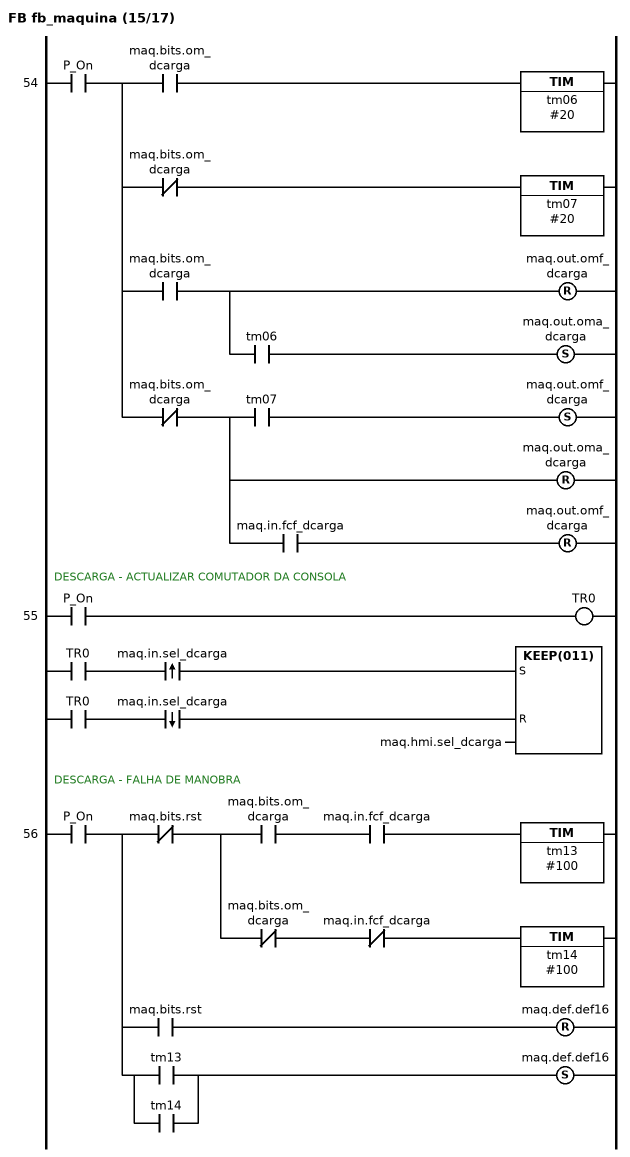
; rung 54
LD P_On
OUT TR0
AND maq.bits.om_dcarga
TIM tm06 #20
LD TR0
ANDNOT maq.bits.om_dcarga
TIM tm07 #20
LD TR0
AND maq.bits.om_dcarga
RSET maq.out.omf_dcarga
AND tm06
SET maq.out.oma_dcarga
LD TR0
ANDNOT maq.bits.om_dcarga
OUT TR1
AND tm07
SET maq.out.omf_dcarga
LD TR1
RSET maq.out.oma_dcarga
AND maq.in.fcf_dcarga
RSET maq.out.omf_dcarga
; rung 55: DESCARGA - ACTUALIZAR COMUTADOR DA CONSOLA
LD P_On
OUT TR0
LD TR0
@AND maq.in.sel_dcarga
LD TR0
%AND maq.in.sel_dcarga
KEEP(011) maq.hmi.sel_dcarga
; rung 56: DESCARGA - FALHA DE MANOBRA
LD P_On
OUT TR0
ANDNOT maq.bits.rst
OUT TR1
AND maq.bits.om_dcarga
AND maq.in.fcf_dcarga
TIM tm13 #100
LD TR1
ANDNOT maq.bits.om_dcarga
ANDNOT maq.in.fcf_dcarga
TIM tm14 #100
LD TR0
AND maq.bits.rst
RSET maq.def.def16
LD TR0
LD tm13
OR tm14
ANDLD
SET maq.def.def16

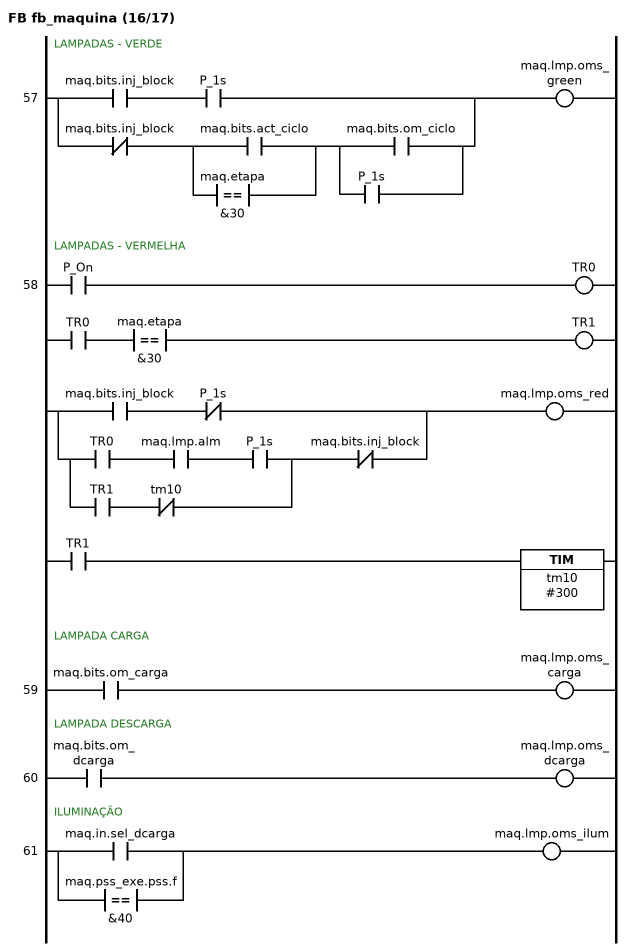
; rung 57: LAMPADAS - VERDE
LD maq.bits.inj_block
AND P_1s
LDNOT maq.bits.inj_block
LD maq.bits.act_ciclo
OR=(300) maq.etapa &30
ANDLD
LD maq.bits.om_ciclo
OR P_1s
ANDLD
ORLD
OUT maq.lmp.oms_green
; rung 58: LAMPADAS - VERMELHA
LD P_On
OUT TR0
LD TR0
AND=(300) maq.etapa &30
OUT TR1
LD maq.bits.inj_block
ANDNOT P_1s
LD TR0
AND maq.lmp.alm
AND P_1s
LD TR1
ANDNOT tm10
ORLD
ANDNOT maq.bits.inj_block
ORLD
OUT maq.lmp.oms_red
LD TR1
TIM tm10 #300
; rung 59: LAMPADA CARGA
LD maq.bits.om_carga
OUT maq.lmp.oms_carga
; rung 60: LAMPADA DESCARGA
LD maq.bits.om_dcarga
OUT maq.lmp.oms_dcarga
; rung 61: ILUMINAÇÃO
LD maq.in.sel_dcarga
OR=(300) maq.pss_exe.pss.f &40
OUT maq.lmp.oms_ilum

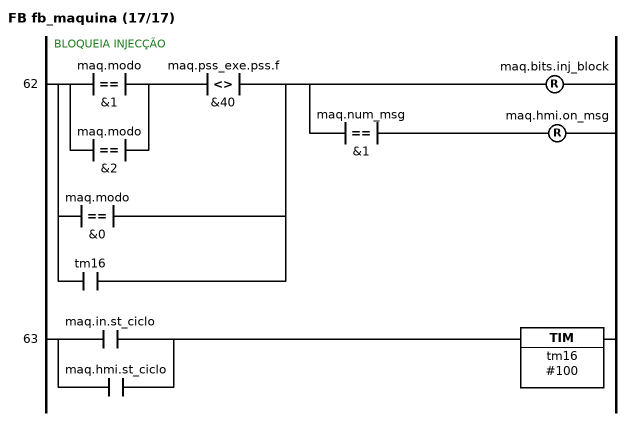
; rung 62: BLOQUEIA INJECÇÃO
LD=(300) maq.modo &1
OR=(300) maq.modo &2
AND<>(305) maq.pss_exe.pss.f &40
OR=(300) maq.modo &0
OR tm16
RSET maq.bits.inj_block
AND=(300) maq.num_msg &1
RSET maq.hmi.on_msg
; rung 63
LD maq.in.st_ciclo
OR maq.hmi.st_ciclo
TIM tm16 #100

## Function block fb_maquina_copy_log
; FUNÇÃO COPIA LOG - Copia os dados do passo actual para disponibilizar para fazer datalogger
VAR_INPUT
  tipo : INT;  (* Tipo de copia: 0 - Copia user/lote e dados a zero / 1 - Copia com ordem a decorrer (não copia user/lote) / 2 - Fim da ordem (Coloca passo 999) / 3 - Ordem descarregada sem execução (Colocar -3 no passo) *)
END_VAR
VAR_IN_OUT
  maq : s_maquina;  (* Dados da maquina *)
  of_exe : s_of;  (* Ordem de fabrico *)
  mes_com : s_mes_com;  (* Dados de comunicação com o MES *)
END_VAR
(*Não executa se ainda não tiver feito o log*)
IF maq.log.pss_exe.log=TRUE THEN
	RETURN;
END_IF;

maq.pss_exe.log:= TRUE;


(*Dados comuns*)
maq.log.user[0]:= mes_com.user[0];
maq.log.user[1]:= mes_com.user[1];
maq.log.user[2]:= mes_com.user[2];
maq.log.user[3]:= mes_com.user[3];
maq.log.user[4]:= mes_com.user[4];
maq.log.user[5]:= mes_com.user[5];
maq.log.user[6]:= mes_com.user[6];
maq.log.user[7]:= mes_com.user[7];
maq.log.user[8]:= mes_com.user[8];
maq.log.user[9]:= mes_com.user[9];
	
maq.log.n_of[0]:= of_exe.cliente.n_lt[0];
maq.log.n_of[1]:= of_exe.cliente.n_lt[1];
maq.log.n_of[2]:= of_exe.cliente.n_lt[2];
maq.log.n_of[3]:= of_exe.cliente.n_lt[3];
maq.log.n_of[4]:= of_exe.cliente.n_lt[4];
maq.log.n_of[5]:= of_exe.cliente.n_lt[5];
maq.log.n_of[6]:= of_exe.cliente.n_lt[6];
maq.log.n_of[7]:= of_exe.cliente.n_lt[7];
maq.log.n_of[8]:= of_exe.cliente.n_lt[8];
maq.log.n_of[9]:= of_exe.cliente.n_lt[9];

maq.log.pss_exe.exc:= maq.pss_exe.exc;
maq.log.pss_exe.exe:= maq.pss_exe.exe;	
maq.log.pss_exe.ini:= maq.pss_exe.ini;	
maq.log.pss_exe.fim:= maq.pss_exe.fim;	
maq.log.pss_exe.log:= maq.pss_exe.log;	

(*Registo inicial*)
IF tipo=0 THEN	
	maq.log.pss_exe.num_pss:= 0;
	maq.log.pss_exe.pss.f:= 0;
	maq.log.pss_exe.pss.p1:= 0;
	maq.log.pss_exe.pss.p2:= 0,0;
	maq.log.pss_exe.pss.tt:= 0,0;
	maq.log.pss_exe.pss.uni:= 0;
END_IF;

(*Ordem em execução*)
IF tipo=1 THEN	
	maq.log.pss_exe.num_pss:= maq.pss_exe.num_pss+1;
	maq.log.pss_exe.pss.f:= maq.pss_exe.pss.f;
	maq.log.pss_exe.pss.p1:= maq.pss_exe.pss.p1;
	maq.log.pss_exe.pss.p2:= maq.pss_exe.pss.p2;
	maq.log.pss_exe.pss.tt:= maq.pss_exe.pss.tt;
	maq.log.pss_exe.pss.uni:= maq.pss_exe.pss.uni;
END_IF;
	
(*Ordem terminada*)	
IF tipo=2 THEN
	maq.log.pss_exe.num_pss:= 999;
	maq.log.pss_exe.pss.f:= 0;
	maq.log.pss_exe.pss.p1:= 0;
	maq.log.pss_exe.pss.p2:= 0,0;
	maq.log.pss_exe.pss.tt:= 0,0;
	maq.log.pss_exe.pss.uni:= 0;
END_IF;	

(*Ordem não executada*)
IF tipo=3 THEN
	maq.log.pss_exe.num_pss:= -3;
	maq.log.pss_exe.pss.f:= 0;
	maq.log.pss_exe.pss.p1:= 0;
	maq.log.pss_exe.pss.p2:= 0,0;
	maq.log.pss_exe.pss.tt:= 0,0;
	maq.log.pss_exe.pss.uni:= 0;	
END_IF;	

## Function block fb_maquina_mov_pss_act
; FUNÇÃO MAQUINA MOVE PASSOS ACTUAIS - Faz a passagem da função do passo actual da maquina para a zona de memoria do passo actual. Faz também a passagem do total do passo em execução.
VAR_IN_OUT
  maq : s_maquina;  (* Dados da maquina *)
  of_exe : s_of;  (* Ordem de fabrico *)
END_VAR
(*Não esta a executar nenhum passo - Limpeza da zona de memória do passo actual*)
	IF maq.pss_exe.num_pss=-1 THEN
		maq.pss_exe.pss.f:= 0;
		maq.pss_exe.pss.p1:= 0;
		maq.pss_exe.pss.p2:=0,0;
		maq.pss_exe.pss.tt:= 0,0;
		maq.pss_exe.pss.uni:= 0;
	END_IF;

(*Leitura do passo actual e passagem dos valores*)
	IF maq.pss_exe.num_pss=0 THEN
		maq.pss_exe.pss.f:= of_exe.prg.pss[0].f;
		maq.pss_exe.pss.p1:= of_exe.prg.pss[0].p1;
		maq.pss_exe.pss.p2:= of_exe.prg.pss[0].p2;
		of_exe.prg.pss[0].tt:= maq.pss_exe.pss.tt;
		maq.pss_exe.pss.uni:=of_exe.prg.pss[0].uni;
	END_IF;

	IF maq.pss_exe.num_pss=1 THEN
		maq.pss_exe.pss.f:= of_exe.prg.pss[1].f;
		maq.pss_exe.pss.p1:= of_exe.prg.pss[1].p1;
		maq.pss_exe.pss.p2:= of_exe.prg.pss[1].p2;
		of_exe.prg.pss[1].tt:= maq.pss_exe.pss.tt;
		maq.pss_exe.pss.uni:=of_exe.prg.pss[1].uni;
	END_IF;

	IF maq.pss_exe.num_pss=2 THEN
		maq.pss_exe.pss.f:= of_exe.prg.pss[2].f;
		maq.pss_exe.pss.p1:= of_exe.prg.pss[2].p1;
		maq.pss_exe.pss.p2:= of_exe.prg.pss[2].p2;
		of_exe.prg.pss[2].tt:= maq.pss_exe.pss.tt;
		maq.pss_exe.pss.uni:=of_exe.prg.pss[2].uni;
	END_IF;

	IF maq.pss_exe.num_pss=3 THEN
		maq.pss_exe.pss.f:= of_exe.prg.pss[3].f;
		maq.pss_exe.pss.p1:= of_exe.prg.pss[3].p1;
		maq.pss_exe.pss.p2:= of_exe.prg.pss[3].p2;
		of_exe.prg.pss[3].tt:= maq.pss_exe.pss.tt;
		maq.pss_exe.pss.uni:=of_exe.prg.pss[3].uni;
	END_IF;

	IF maq.pss_exe.num_pss=4 THEN
		maq.pss_exe.pss.f:= of_exe.prg.pss[4].f;
		maq.pss_exe.pss.p1:= of_exe.prg.pss[4].p1;
		maq.pss_exe.pss.p2:= of_exe.prg.pss[4].p2;
		of_exe.prg.pss[4].tt:= maq.pss_exe.pss.tt;
		maq.pss_exe.pss.uni:=of_exe.prg.pss[4].uni;
	END_IF;

	IF maq.pss_exe.num_pss=5 THEN
		maq.pss_exe.pss.f:= of_exe.prg.pss[5].f;
		maq.pss_exe.pss.p1:= of_exe.prg.pss[5].p1;
		maq.pss_exe.pss.p2:= of_exe.prg.pss[5].p2;
		of_exe.prg.pss[5].tt:= maq.pss_exe.pss.tt;
		maq.pss_exe.pss.uni:=of_exe.prg.pss[5].uni;
	END_IF;

	IF maq.pss_exe.num_pss=6 THEN
		maq.pss_exe.pss.f:= of_exe.prg.pss[6].f;
		maq.pss_exe.pss.p1:= of_exe.prg.pss[6].p1;
		maq.pss_exe.pss.p2:= of_exe.prg.pss[6].p2;
		of_exe.prg.pss[6].tt:= maq.pss_exe.pss.tt;
		maq.pss_exe.pss.uni:=of_exe.prg.pss[6].uni;
	END_IF;

	IF maq.pss_exe.num_pss=7 THEN
		maq.pss_exe.pss.f:= of_exe.prg.pss[7].f;
		maq.pss_exe.pss.p1:= of_exe.prg.pss[7].p1;
		maq.pss_exe.pss.p2:= of_exe.prg.pss[7].p2;
		of_exe.prg.pss[7].tt:= maq.pss_exe.pss.tt;
		maq.pss_exe.pss.uni:=of_exe.prg.pss[7].uni;
	END_IF;

	IF maq.pss_exe.num_pss=8 THEN
		maq.pss_exe.pss.f:= of_exe.prg.pss[8].f;
		maq.pss_exe.pss.p1:= of_exe.prg.pss[8].p1;
		maq.pss_exe.pss.p2:= of_exe.prg.pss[8].p2;
		of_exe.prg.pss[8].tt:= maq.pss_exe.pss.tt;
		maq.pss_exe.pss.uni:=of_exe.prg.pss[8].uni;
	END_IF;

	IF maq.pss_exe.num_pss=9 THEN
		maq.pss_exe.pss.f:= of_exe.prg.pss[9].f;
		maq.pss_exe.pss.p1:= of_exe.prg.pss[9].p1;
		maq.pss_exe.pss.p2:= of_exe.prg.pss[9].p2;
		of_exe.prg.pss[9].tt:= maq.pss_exe.pss.tt;
		maq.pss_exe.pss.uni:=of_exe.prg.pss[9].uni;
	END_IF;

	IF maq.pss_exe.num_pss=10 THEN
		maq.pss_exe.pss.f:= of_exe.prg.pss[10].f;
		maq.pss_exe.pss.p1:= of_exe.prg.pss[10].p1;
		maq.pss_exe.pss.p2:= of_exe.prg.pss[10].p2;
		of_exe.prg.pss[10].tt:= maq.pss_exe.pss.tt;
		maq.pss_exe.pss.uni:=of_exe.prg.pss[10].uni;
	END_IF;

	IF maq.pss_exe.num_pss=11 THEN
		maq.pss_exe.pss.f:= of_exe.prg.pss[11].f;
		maq.pss_exe.pss.p1:= of_exe.prg.pss[11].p1;
		maq.pss_exe.pss.p2:= of_exe.prg.pss[11].p2;
		of_exe.prg.pss[11].tt:= maq.pss_exe.pss.tt;
		maq.pss_exe.pss.uni:=of_exe.prg.pss[11].uni;
	END_IF;

## Function block fb_maquina_pss_2_str10_PT
; FUNÇÃO PASSO PARA STRING - Transforma os passo em execução em strings para apresentar no HMI.
VAR_IN_OUT
  prg : s_of_prg;  (* Programa *)
  str_pss0 : STRING;  (* String do passo *)
  str_pss1 : STRING;  (* String do passo *)
  str_pss2 : STRING;  (* String do passo *)
  str_pss3 : STRING;  (* String do passo *)
  str_pss4 : STRING;  (* String do passo *)
  str_pss5 : STRING;  (* String do passo *)
  str_pss6 : STRING;  (* String do passo *)
  str_pss7 : STRING;  (* String do passo *)
  str_pss8 : STRING;  (* String do passo *)
  str_pss9 : STRING;  (* String do passo *)
  str_pss10 : STRING;
  str_pss11 : STRING;
  maq : s_maquina;  (* Dados da maquina *)
  str_act : STRING;  (* String do passo actual *)
END_VAR
VAR
  str_p1 : STRING;  (* Parametro 1 *)
  str_p2 : STRING;  (* Parametro 2 *)
  dd : REAL;  (* Dividendo *)
  dv : REAL;  (* Divisor *)
  qc : REAL;  (* Quociente *)
  r : REAL;  (* Resto *)
  i : INT;
  pss : s_of_pss;  (* Passo *)
  str_pss : STRING;  (* String do passo *)
END_VAR
FOR i:= 0 TO 11 DO
	(*Passagem dos dados dos varios passos*)
	CASE i OF
		0:	pss.f:= prg.pss[0].f;pss.p1:= prg.pss[0].p1;pss.p2:=prg.pss[0].p2;
		1:	pss.f:= prg.pss[1].f;pss.p1:= prg.pss[1].p1;pss.p2:=prg.pss[1].p2;
		2:	pss.f:= prg.pss[2].f;pss.p1:= prg.pss[2].p1;pss.p2:=prg.pss[2].p2;
		3:	pss.f:= prg.pss[3].f;pss.p1:= prg.pss[3].p1;pss.p2:=prg.pss[3].p2;
		4:	pss.f:= prg.pss[4].f;pss.p1:= prg.pss[4].p1;pss.p2:=prg.pss[4].p2;
		5:	pss.f:= prg.pss[5].f;pss.p1:= prg.pss[5].p1;pss.p2:=prg.pss[5].p2;
		6:	pss.f:= prg.pss[6].f;pss.p1:= prg.pss[6].p1;pss.p2:=prg.pss[6].p2;
		7:	pss.f:= prg.pss[7].f;pss.p1:= prg.pss[7].p1;pss.p2:=prg.pss[7].p2;
		8:	pss.f:= prg.pss[8].f;pss.p1:= prg.pss[8].p1;pss.p2:=prg.pss[8].p2;
		9:	pss.f:= prg.pss[9].f;pss.p1:= prg.pss[9].p1;pss.p2:=prg.pss[9].p2;
		10:	pss.f:= prg.pss[10].f;pss.p1:= prg.pss[10].p1;pss.p2:=prg.pss[10].p2;
		11:	pss.f:= prg.pss[11].f;pss.p1:= prg.pss[11].p1;pss.p2:=prg.pss[11].p2;
	END_CASE;
	(*Inicialização*)
		str_pss:= '';
 
 	(*Transformação dos valores em string*)
	 str_p1:= INT_TO_STRING(pss.p1);
 
 	dd:= pss.p2*10,0;
 	dv:= 10,0;
 	qc:=INT_TO_REAL(REAL_TO_INT(dd/dv));
 	r:= dd-dv*qc;
	IF r<0,0 THEN
		qc:= qc-1,0;
		r:= 10,0+r;
	END_IF;
	
 	str_p2:= CONCAT(INT_TO_STRING(REAL_TO_INT(qc)),',',INT_TO_STRING(REAL_TO_INT(r)));

  	(*Aspiração*)
 	IF pss.f=10 THEN
		 str_pss:=CONCAT('Aspirazione ',str_p1,'s');
	END_IF;

	(*Aquecimento*)
 	IF pss.f=20 THEN
		 str_pss:=CONCAT('Riscaldamento ',str_p2,'ºC ',str_p1,'s');
	END_IF;

  	(*Tratamento*)
 	IF pss.f=30 THEN
		 str_pss:=CONCAT('Trattamento ',str_p1,'s');
	END_IF;

  	(*Injecção*)
 	IF pss.f=40 THEN
		 CASE pss.p1 OF
		 	1:str_pss:=CONCAT('BOPSIL ',str_p2,'ml');  (*BOPSIL*)
			2:str_pss:=CONCAT('P28 ',str_p2,'ml');  (*P28*)
			3:str_pss:=CONCAT('SILBIONE ',str_p2,'ml');  (*SILICONE*)
			4:str_pss:=CONCAT('P2X ',str_p2,'ml');  (*P2X*)
			5:str_pss:=CONCAT('LC104 ',str_p2,'ml');  (*LC104*)
			6:str_pss:=CONCAT('PARAFFINA ',str_p2,'ml');  (*PARAFINA*)
			7:str_pss:=CONCAT('TEFLON ',str_p2,'ml');  (*TEFLON*)
			8:str_pss:=CONCAT('CAF ',str_p2,'ml');  (*CAF*)
			9:str_pss:=CONCAT('X15 ',str_p2,'ml');  (*X15*)
			10:str_pss:=CONCAT('SWAM P.N.S. ',str_p2,'ml');  (*SWAM P.N.S.*)
			11:str_pss:=CONCAT('SWAM P.SA ',str_p2,'ml');  (*SWAM P.SA*)		
			19:str_pss:=CONCAT('TR02 ',str_p2,'ml');  (*TR02*)
		END_CASE;
	END_IF;

  	(*LOAD*)
 	IF pss.f=70 THEN
		 str_pss:='Carico ';
	END_IF;

  	(*UNLOAD*)
 	IF pss.f=80 THEN
		 str_pss:='Scarico ';
	END_IF;
	
	(*Passagem das strings dos varios passos*)
	CASE i OF
		0:	str_pss0:= str_pss;
		1:	str_pss1:= str_pss;
		2:	str_pss2:= str_pss;
		3:	str_pss3:= str_pss;
		4:	str_pss4:= str_pss;
		5:	str_pss5:= str_pss;
		6:	str_pss6:= str_pss;
		7:	str_pss7:= str_pss;
		8:	str_pss8:= str_pss;
		9:	str_pss9:= str_pss;
		10:	str_pss10:= str_pss;
		11:	str_pss11:= str_pss;
	END_CASE;
	
	(*String do passo actual*)
	str_act:= '';
	CASE maq.pss_exe.num_pss OF
		0:	str_act:= str_pss0;
		1:	str_act:= str_pss1;
		2:	str_act:= str_pss2;
		3:	str_act:= str_pss3;
		4:	str_act:= str_pss4;
		5:	str_act:= str_pss5;
		6:	str_act:= str_pss6;
		7:	str_act:= str_pss7;
		8:	str_act:= str_pss8;
		9:	str_act:= str_pss9;
		10:	str_act:= str_pss10;
		11:	str_act:= str_pss11;
	END_CASE;
		
END_FOR;

## Function block fb_mes_com_exe
; COMUNICAÇÃO COM O MES - FUNÇÃO ARRANQUE DE ORDEM - Faz o controlo de comunicação do inicio de ordem com o MES
VAR_IN_OUT
  mes_com : s_mes_com;  (* Dados de comunicação com o MES *)
  of_exe : s_of;  (* Dados da ordem de fabrico a ser executada *)
END_VAR
VAR
  tm01 : TIMER;
  tm01_st : BOOL;
  mmss AT A351 : INT;
END_VAR
(*Falha de comunicação*)

tm01_st:=( mes_com.mes_plc =  mes_com.mes_plcx);
TIMX(tm01_st,tm01,600);
mes_com.mes_com_fail:= tm01.CF;

mes_com.mes_plcx:= mes_com.mes_plc;

(*Variável de comunicação para o MES*)
mes_com.plc_mes:= mmss;

(*FUNÇÕES
	0 - Nada
	1- Inicio de ordem
	2 - Fim de ordem
	3 - Cancela
	4 - Descarga sem tratamento
	*)
	
(*ESTADOS:
	0 - Nada
	1- Espera dados do MES
	2 - Inicio OK 
	3 - Fim OK
	4 - Erro de OF
	5 - Erro de user
	6 - Erro de comunicação*)

(* Função 0 - NADA*)

(* Função 1 - INICIO OF*)
IF mes_com.f_in_exe=1 AND (mes_com.ctrl_com_mes=0 OR mes_com.f_out_exe=1) THEN
	IF mes_com.f_out_exe=0 THEN

		mes_com.n_enc[0]:= of_exe.cliente.n_enc[0];
		mes_com.n_enc[1]:= of_exe.cliente.n_enc[1];
		mes_com.n_enc[2]:= of_exe.cliente.n_enc[2];
		mes_com.n_enc[3]:= of_exe.cliente.n_enc[3];
		mes_com.n_enc[4]:= of_exe.cliente.n_enc[4];
		mes_com.n_enc[5]:= of_exe.cliente.n_enc[5];
		mes_com.n_enc[6]:= of_exe.cliente.n_enc[6];
		mes_com.n_enc[7]:= of_exe.cliente.n_enc[7];
		mes_com.n_enc[8]:= of_exe.cliente.n_enc[8];
		mes_com.n_enc[9]:= of_exe.cliente.n_enc[9];

		mes_com.n_of[0]:= of_exe.cliente.n_of[0];
		mes_com.n_of[1]:= of_exe.cliente.n_of[1];
		mes_com.n_of[2]:= of_exe.cliente.n_of[2];
		mes_com.n_of[3]:= of_exe.cliente.n_of[3];
		mes_com.n_of[4]:= of_exe.cliente.n_of[4];
		mes_com.n_of[5]:= of_exe.cliente.n_of[5];
		mes_com.n_of[6]:= of_exe.cliente.n_of[6];
		mes_com.n_of[7]:= of_exe.cliente.n_of[7];
		mes_com.n_of[8]:= of_exe.cliente.n_of[8];
		mes_com.n_of[9]:= of_exe.cliente.n_of[9];		
		
		mes_com.n_lt[0]:= of_exe.cliente.n_lt[0];
		mes_com.n_lt[1]:= of_exe.cliente.n_lt[1];
		mes_com.n_lt[2]:= of_exe.cliente.n_lt[2];
		mes_com.n_lt[3]:= of_exe.cliente.n_lt[3];
		mes_com.n_lt[4]:= of_exe.cliente.n_lt[4];
		mes_com.n_lt[5]:= of_exe.cliente.n_lt[5];
		mes_com.n_lt[6]:= of_exe.cliente.n_lt[6];
		mes_com.n_lt[7]:= of_exe.cliente.n_lt[7];
		mes_com.n_lt[8]:= of_exe.cliente.n_lt[8];
		mes_com.n_lt[9]:= of_exe.cliente.n_lt[9];		
		
		mes_com.ctrl_com_plc:= -4;
		mes_com.new_of:= mes_com.new_of+1;
		IF mes_com.new_of>10000 OR mes_com.new_of<0 THEN
			mes_com.new_of:= 0;
		END_IF;		
	END_IF;
	mes_com.f_out_exe:= 1;
		(*MES OK - INICIO DE ORDEM*)
	IF mes_com.ctrl_com_mes=4 THEN
		mes_com.f_out_exe:= 2;
		 mes_com.f_in_exe:= 0;
		mes_com.ctrl_com_plc:= 0;		 
	END_IF;
		(*MES NOK - Mostra erro*)
	IF mes_com.ctrl_com_mes=101 THEN
		mes_com.f_out_exe:= 4;
		mes_com.f_in_exe:= 0;
		mes_com.ctrl_com_plc:= 0;		 
	END_IF;
	IF mes_com.ctrl_com_mes=102 THEN
		mes_com.f_out_exe:= 5;
		mes_com.f_in_exe:= 0;
		mes_com.ctrl_com_plc:= 0;		 
	END_IF;
END_IF;

(* Função 2 - FIM OF*)
IF mes_com.f_in_exe=2 THEN
	mes_com.ctrl_com_plc:= -5;	
	
	mes_com.f_out_exe:= 1;	
		(*MES OK - Ordem terminada*)
	IF mes_com.ctrl_com_mes=5 THEN
		mes_com.f_out_exe:= 3;
		 mes_com.f_in_exe:= 3;
		 mes_com.ctrl_com_plc:= 0;
	END_IF;
		(*MES NOK - Mostra erro*)
	IF mes_com.ctrl_com_mes=101 THEN
		mes_com.f_out_exe:= 4;
		mes_com.f_in_exe:= 3;
		mes_com.ctrl_com_plc:= 0;		 
	END_IF;
	IF mes_com.ctrl_com_mes=102 THEN
		mes_com.f_out_exe:= 5;
		mes_com.f_in_exe:= 3;
		mes_com.ctrl_com_plc:= 0;		 
	END_IF;	
END_IF;

(* Função 3 - CANCELA*)
IF mes_com.f_in_exe=3 THEN
	
	mes_com.ctrl_com_plc:= 0;
	mes_com.f_out_exe:= 0;
	mes_com.f_in_exe:= 0;
	
	mes_com.n_enc[0]:= 0;
	mes_com.n_enc[1]:= 0;
	mes_com.n_enc[2]:= 0;
	mes_com.n_enc[3]:= 0;
	mes_com.n_enc[4]:= 0;
	mes_com.n_enc[5]:= 0;
	mes_com.n_enc[6]:= 0;
	mes_com.n_enc[7]:= 0;
	mes_com.n_enc[8]:= 0;
	mes_com.n_enc[9]:= 0;
	
	mes_com.n_of[0]:= 0;
	mes_com.n_of[1]:= 0;
	mes_com.n_of[2]:= 0;
	mes_com.n_of[3]:= 0;
	mes_com.n_of[4]:= 0;
	mes_com.n_of[5]:= 0;
	mes_com.n_of[6]:= 0;
	mes_com.n_of[7]:= 0;
	mes_com.n_of[8]:= 0;
	mes_com.n_of[9]:= 0;
	
	mes_com.n_lt[0]:= 0;
	mes_com.n_lt[1]:= 0;
	mes_com.n_lt[2]:= 0;
	mes_com.n_lt[3]:= 0;
	mes_com.n_lt[4]:= 0;
	mes_com.n_lt[5]:= 0;
	mes_com.n_lt[6]:= 0;
	mes_com.n_lt[7]:= 0;
	mes_com.n_lt[8]:= 0;
	mes_com.n_lt[9]:= 0;	
		
END_IF;

(* Função 4 - DESCARGA SEM TRATAMENTO*)
IF mes_com.f_in_exe=4 THEN
		mes_com.ctrl_com_plc:= -3;

		mes_com.n_enc[0]:= of_exe.cliente.n_enc[0];
		mes_com.n_enc[1]:= of_exe.cliente.n_enc[1];
		mes_com.n_enc[2]:= of_exe.cliente.n_enc[2];
		mes_com.n_enc[3]:= of_exe.cliente.n_enc[3];
		mes_com.n_enc[4]:= of_exe.cliente.n_enc[4];
		mes_com.n_enc[5]:= of_exe.cliente.n_enc[5];
		mes_com.n_enc[6]:= of_exe.cliente.n_enc[6];
		mes_com.n_enc[7]:= of_exe.cliente.n_enc[7];
		mes_com.n_enc[8]:= of_exe.cliente.n_enc[8];
		mes_com.n_enc[9]:= of_exe.cliente.n_enc[9];

		mes_com.n_of[0]:= of_exe.cliente.n_of[0];
		mes_com.n_of[1]:= of_exe.cliente.n_of[1];
		mes_com.n_of[2]:= of_exe.cliente.n_of[2];
		mes_com.n_of[3]:= of_exe.cliente.n_of[3];
		mes_com.n_of[4]:= of_exe.cliente.n_of[4];
		mes_com.n_of[5]:= of_exe.cliente.n_of[5];
		mes_com.n_of[6]:= of_exe.cliente.n_of[6];
		mes_com.n_of[7]:= of_exe.cliente.n_of[7];
		mes_com.n_of[8]:= of_exe.cliente.n_of[8];
		mes_com.n_of[9]:= of_exe.cliente.n_of[9];		
		
		mes_com.n_lt[0]:= of_exe.cliente.n_lt[0];
		mes_com.n_lt[1]:= of_exe.cliente.n_lt[1];
		mes_com.n_lt[2]:= of_exe.cliente.n_lt[2];
		mes_com.n_lt[3]:= of_exe.cliente.n_lt[3];
		mes_com.n_lt[4]:= of_exe.cliente.n_lt[4];
		mes_com.n_lt[5]:= of_exe.cliente.n_lt[5];
		mes_com.n_lt[6]:= of_exe.cliente.n_lt[6];
		mes_com.n_lt[7]:= of_exe.cliente.n_lt[7];
		mes_com.n_lt[8]:= of_exe.cliente.n_lt[8];
		mes_com.n_lt[9]:= of_exe.cliente.n_lt[9];		
	
	mes_com.f_out_exe:= 1;	
		(*MES OK - Ordem terminada*)
	IF mes_com.ctrl_com_mes=3 THEN
		mes_com.f_out_exe:= 3;
		 mes_com.f_in_exe:= 3;
		 mes_com.ctrl_com_plc:= 0;
	END_IF;
		(*MES NOK - Mostra erro*)
	IF mes_com.ctrl_com_mes=101 THEN
		mes_com.f_out_exe:= 4;
		mes_com.f_in_exe:= 3;
		mes_com.ctrl_com_plc:= 0;		 
	END_IF;
	IF mes_com.ctrl_com_mes=102 THEN
		mes_com.f_out_exe:= 5;
		mes_com.f_in_exe:= 3;
		mes_com.ctrl_com_plc:= 0;		 
	END_IF;	
END_IF;
	
(*Falha de comunicação - Mostra janela de falha de comunicação*)
IF mes_com.mes_com_fail=TRUE THEN
	mes_com.f_out_exe:= 6;
	mes_com.f_in_exe:= 0;
	
	mes_com.ctrl_com_plc:= 0;
 	mes_com.ctrl_com_mes:= 0;		
END_IF;
IF  mes_com.mes_com_fail=FALSE AND mes_com.f_out_exe= 6 THEN
	mes_com.f_out_exe:= 0;
END_IF;

## Function block fb_mes_com_trp
; COMUNICAÇÃO COM O MES - FUNÇÃO TRANSPORTE - Faz o controlo de comunicação do transporte com o MES
VAR_INPUT
  ok_trp : BOOL;  (* Transporte OK *)
  ndp_trp : BOOL;  (* Transporte OK *)
END_VAR
VAR_IN_OUT
  mes_com : s_mes_com;  (* Dados de comunicação com o MES *)
  of_mes : s_of;  (* Dados da ordem de fabrico vindos do MES *)
  of_trp : s_of;  (* Dados da ordem de fabrico para o transporte *)
END_VAR
VAR
  tm01 : TIMER;
  tm02 : TIMER;
  tm01_st : BOOL;
  fb_of_clear : fb_of_clear;
  fb_of_copy : fb_of_copy;
  mmss AT A351 : INT;
  com_step : INT;
END_VAR
(*Falha de comunicação*)
tm01_st:=( mes_com.mes_plc =  mes_com.mes_plcx);
TIMX(tm01_st,tm01,600);
mes_com.mes_com_fail:= tm01.CF;

mes_com.mes_plcx:= mes_com.mes_plc;

(*Variável de comunicação para o MES*)
mes_com.plc_mes:= mmss;

(*FUNÇÕES
	0 - Nada
	1 - Pede info de OF
	2 - Transporta online
	3 - Cancela
	4 - Pede transporte offline
	5 - Transporta offline
	6 - Pede transporte online
	*)
	
(*ESTADOS:
	0 - Janela de introdução user/OF
	1 - Espera dados do MES
	2 - Janela de info de OF
	3 - Janela de transporte
	4 - Erro de OF
	5 - Erro de user
	6 - Erro de comunicação
	7 - Transporte manual
	8 - Transporte indisponivel
	9 - Maquina carregada
	10 - Ordem já alocada
	11 - Lote pertence à ordem actual*)

(* Função 0 - NADA*)

(* Função 1 - PEDE INFO DE OF*)
IF mes_com.f_in_exe=1 THEN
	IF com_step=0 AND  mes_com.ctrl_com_mes=0 THEN
		com_step:= 1;
	END_IF;
	
	IF com_step=1 THEN
		mes_com.ctrl_com_plc:= -1;
		mes_com.new_of:= mes_com.new_of+1;
		IF mes_com.new_of>10000 OR mes_com.new_of<0 THEN
			mes_com.new_of:= 0;
		END_IF;
		com_step:= 2;
	END_IF;
	mes_com.f_out_exe:= 1;
	IF com_step= 2 THEN
		(*MES OK - Mostra info da OF*)
		IF mes_com.ctrl_com_mes=1 THEN
			mes_com.f_out_exe:= 2;
			 mes_com.f_in_exe:= 0;
			 mes_com.ctrl_com_plc:= 0;
		END_IF;
			(*MES NOK - Mostra erro*)
		IF mes_com.ctrl_com_mes=101 THEN
			mes_com.f_out_exe:= 4;
			mes_com.f_in_exe:= 0;
			mes_com.ctrl_com_plc:= 0;
		END_IF;
		IF mes_com.ctrl_com_mes=102 THEN
			mes_com.f_out_exe:= 5;
			mes_com.f_in_exe:= 0;
			mes_com.ctrl_com_plc:= 0;
		END_IF;
		IF mes_com.ctrl_com_mes=103 THEN
			mes_com.f_out_exe:= 10;
			mes_com.f_in_exe:= 0;
			mes_com.ctrl_com_plc:= 0;
		END_IF;
		IF mes_com.ctrl_com_mes=104 THEN
			mes_com.f_out_exe:= 11;
			mes_com.f_in_exe:= 0;
			mes_com.ctrl_com_plc:= 0;
		END_IF;	
	END_IF;
END_IF;

(* Função 2 - TRANSPORTA*)
IF mes_com.f_in_exe=2 AND NOT of_trp.dados THEN
	IF mes_com.f_out_exe=2 THEN
		of_mes.dados:= TRUE;
		of_mes.online:= TRUE;
		fb_of_copy(of_mes,of_trp);
		mes_com.f_out_exe:= 3;
		 mes_com.f_in_exe:= 0;
		 mes_com.ctrl_com_plc:= 0;
	END_IF;	
END_IF;

(* Função 3 - CANCELA*)
IF mes_com.f_in_exe=3 THEN
	of_mes.dados:= FALSE;
	
	mes_com.ctrl_com_plc:= 0;
	com_step:= 0;
	mes_com.f_out_exe:= 0;
	mes_com.f_in_exe:= 0;
	
	mes_com.n_enc[0]:= 0;
	mes_com.n_enc[1]:= 0;
	mes_com.n_enc[2]:= 0;
	mes_com.n_enc[3]:= 0;
	mes_com.n_enc[4]:= 0;
	mes_com.n_enc[5]:= 0;
	mes_com.n_enc[6]:= 0;
	mes_com.n_enc[7]:= 0;
	mes_com.n_enc[8]:= 0;
	mes_com.n_enc[9]:= 0;
	
	mes_com.n_of[0]:= 0;
	mes_com.n_of[1]:= 0;
	mes_com.n_of[2]:= 0;
	mes_com.n_of[3]:= 0;
	mes_com.n_of[4]:= 0;
	mes_com.n_of[5]:= 0;
	mes_com.n_of[6]:= 0;
	mes_com.n_of[7]:= 0;
	mes_com.n_of[8]:= 0;
	mes_com.n_of[9]:= 0;
	
	mes_com.n_lt[0]:= 0;
	mes_com.n_lt[1]:= 0;
	mes_com.n_lt[2]:= 0;
	mes_com.n_lt[3]:= 0;
	mes_com.n_lt[4]:= 0;
	mes_com.n_lt[5]:= 0;
	mes_com.n_lt[6]:= 0;
	mes_com.n_lt[7]:= 0;
	mes_com.n_lt[8]:= 0;
	mes_com.n_lt[9]:= 0;	
	
	mes_com.user[0]:= 0;
	mes_com.user[1]:= 0;
	mes_com.user[2]:= 0;
	mes_com.user[3]:= 0;
	mes_com.user[4]:= 0;
	mes_com.user[5]:= 0;
	mes_com.user[6]:= 0;
	mes_com.user[7]:= 0;
	mes_com.user[8]:= 0;
	mes_com.user[9]:= 0;		
END_IF;

(*Pede transporte offline*)
IF mes_com.f_in_exe=4 THEN
	mes_com.f_out_exe:= 7;
	mes_com.f_in_exe:= 0;
	mes_com.ctrl_com_plc:= 0;	
END_IF;

(*Transporta offline*)
IF mes_com.f_in_exe=5 AND NOT of_trp.dados THEN
	of_mes.cliente.n_enc[0]:=  mes_com.n_enc[0];
	of_mes.cliente.n_enc[1]:=  mes_com.n_enc[1];
	of_mes.cliente.n_enc[2]:=  mes_com.n_enc[2];
	of_mes.cliente.n_enc[3]:=  mes_com.n_enc[3];
	of_mes.cliente.n_enc[4]:=  mes_com.n_enc[4];
	of_mes.cliente.n_enc[5]:=  mes_com.n_enc[5];
	of_mes.cliente.n_enc[6]:=  mes_com.n_enc[6];
	of_mes.cliente.n_enc[7]:=  mes_com.n_enc[7];
	of_mes.cliente.n_enc[8]:=  mes_com.n_enc[8];
	of_mes.cliente.n_enc[9]:=  mes_com.n_enc[9];
	
	of_mes.cliente.n_of[0]:=  mes_com.n_of[0];
	of_mes.cliente.n_of[1]:=  mes_com.n_of[1];
	of_mes.cliente.n_of[2]:=  mes_com.n_of[2];
	of_mes.cliente.n_of[3]:=  mes_com.n_of[3];
	of_mes.cliente.n_of[4]:=  mes_com.n_of[4];
	of_mes.cliente.n_of[5]:=  mes_com.n_of[5];
	of_mes.cliente.n_of[6]:=  mes_com.n_of[6];
	of_mes.cliente.n_of[7]:=  mes_com.n_of[7];
	of_mes.cliente.n_of[8]:=  mes_com.n_of[8];
	of_mes.cliente.n_of[9]:=  mes_com.n_of[9];
	
	of_mes.cliente.n_lt[0]:=  mes_com.n_lt[0];
	of_mes.cliente.n_lt[1]:=  mes_com.n_lt[1];
	of_mes.cliente.n_lt[2]:=  mes_com.n_lt[2];
	of_mes.cliente.n_lt[3]:=  mes_com.n_lt[3];
	of_mes.cliente.n_lt[4]:=  mes_com.n_lt[4];
	of_mes.cliente.n_lt[5]:=  mes_com.n_lt[5];
	of_mes.cliente.n_lt[6]:=  mes_com.n_lt[6];
	of_mes.cliente.n_lt[7]:=  mes_com.n_lt[7];
	of_mes.cliente.n_lt[8]:=  mes_com.n_lt[8];
	of_mes.cliente.n_lt[9]:=  mes_com.n_lt[9];	
	
	of_mes.dados:= TRUE;
	of_mes.online:= TRUE;
	fb_of_copy(of_mes,of_trp);
	mes_com.f_out_exe:= 3;
	 mes_com.f_in_exe:= 0;
	 mes_com.ctrl_com_plc:= 0;
END_IF;
	
(*Pede transporte online*)
IF mes_com.f_in_exe=6 THEN
	mes_com.f_out_exe:= 0;
	mes_com.f_in_exe:= 0;
	mes_com.ctrl_com_plc:= 0;
END_IF;	
	
IF  mes_com.mes_com_fail=FALSE AND mes_com.f_out_exe= 6 THEN
	mes_com.f_out_exe:= 0;
END_IF;

(*Transporte indisponivel*)
IF ok_trp=FALSE AND ( mes_com.f_out_exe= 0 OR  mes_com.f_out_exe= 7) THEN
	mes_com.f_out_exe:= 8;
	mes_com.f_in_exe:= 0;
END_IF;

IF ok_trp=TRUE AND mes_com.f_out_exe=8 THEN
	mes_com.f_out_exe:= 0;
END_IF;

(*Maquina carregada*)
IF of_trp.dados=TRUE AND ( mes_com.f_out_exe= 0 OR  mes_com.f_out_exe= 7) THEN
	mes_com.f_out_exe:= 9;
	mes_com.f_in_exe:= 0;
END_IF;
IF of_trp.dados=FALSE AND mes_com.f_out_exe=9 THEN
	mes_com.f_out_exe:= 0;
END_IF;

(*Transporte indisponivel*)
IF ndp_trp=TRUE AND ( mes_com.f_out_exe= 0 OR  mes_com.f_out_exe= 7) THEN
	mes_com.f_out_exe:= 12;
	mes_com.f_in_exe:= 0;
END_IF;

IF ndp_trp=FALSE AND mes_com.f_out_exe=12 THEN
	mes_com.f_out_exe:= 0;
END_IF;

(*Falha de comunicação - Mostra janela de falha de comunicação*)
IF mes_com.mes_com_fail=TRUE AND ( mes_com.f_out_exe=0  OR mes_com.f_out_exe=1) THEN
	mes_com.f_out_exe:= 6;
	mes_com.f_in_exe:= 0;
	
	mes_com.ctrl_com_plc:= 0;
 	mes_com.ctrl_com_mes:= 0;			
END_IF;
		
(*Termina ordem de transporte*)
IF mes_com.f_out_exe=3 and ndp_trp=TRUE THEN
	mes_com.f_in_exe:= 3;
END_IF;	

(*Novo pedido*)
IF mes_com.ctrl_com_plc=0 THEN
	com_step:= 0;
END_IF;

## Function block fb_mes_cparagem
; CAUSAS DE PARAGEM - Causas de paragem para o MES
VAR_IN_OUT
  maq : s_maquina;  (* Dados da maquina *)
END_VAR

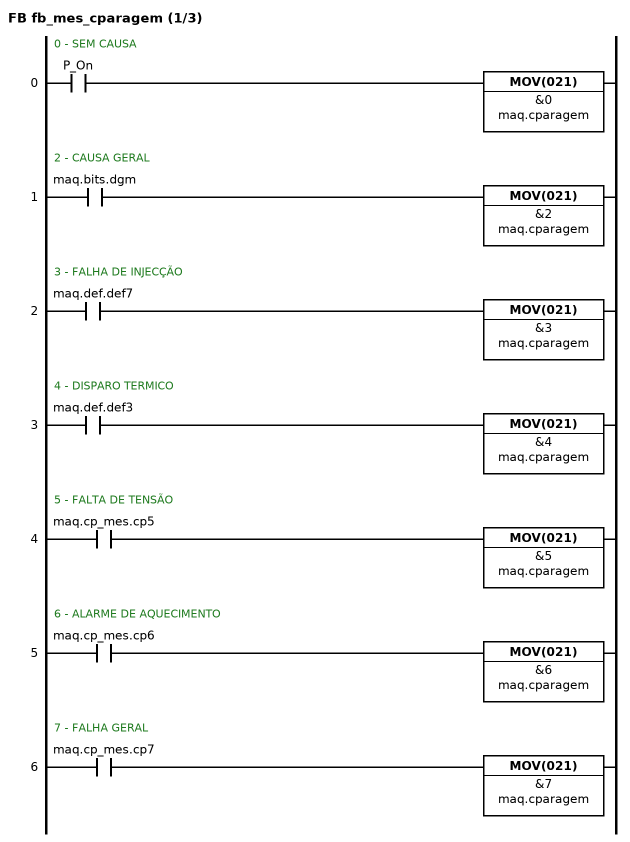
; rung 0: 0 - SEM CAUSA
LD P_On
MOV(021) &0 maq.cparagem
; rung 1: 2 - CAUSA GERAL
LD maq.bits.dgm
MOV(021) &2 maq.cparagem
; rung 2: 3 - FALHA DE INJECÇÃO
LD maq.def.def7
MOV(021) &3 maq.cparagem
; rung 3: 4 - DISPARO TERMICO
LD maq.def.def3
MOV(021) &4 maq.cparagem
; rung 4: 5 - FALTA DE TENSÃO
LD maq.cp_mes.cp5
MOV(021) &5 maq.cparagem
; rung 5: 6 - ALARME DE AQUECIMENTO
LD maq.cp_mes.cp6
MOV(021) &6 maq.cparagem
; rung 6: 7 - FALHA GERAL
LD maq.cp_mes.cp7
MOV(021) &7 maq.cparagem

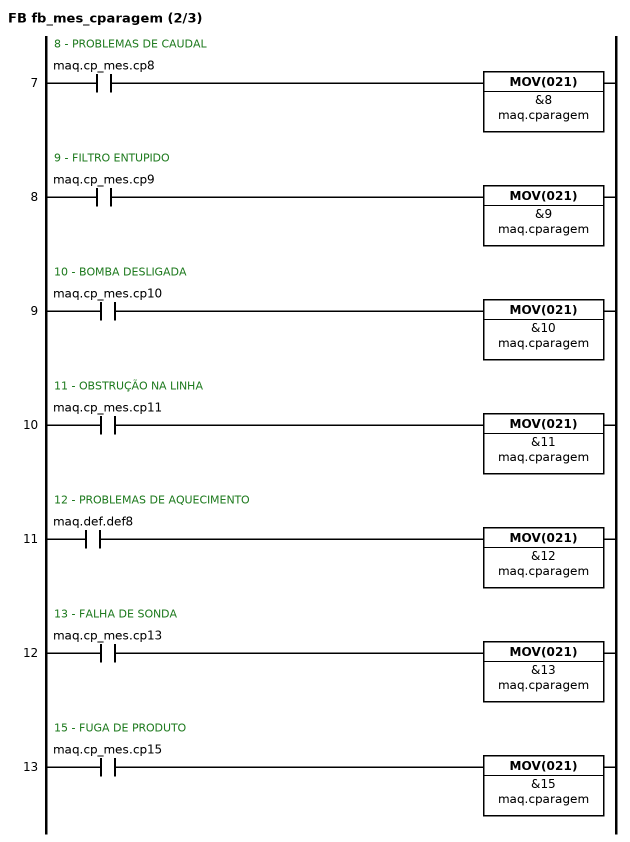
; rung 7: 8 - PROBLEMAS DE CAUDAL
LD maq.cp_mes.cp8
MOV(021) &8 maq.cparagem
; rung 8: 9 - FILTRO ENTUPIDO
LD maq.cp_mes.cp9
MOV(021) &9 maq.cparagem
; rung 9: 10 - BOMBA DESLIGADA
LD maq.cp_mes.cp10
MOV(021) &10 maq.cparagem
; rung 10: 11 - OBSTRUÇÃO NA LINHA
LD maq.cp_mes.cp11
MOV(021) &11 maq.cparagem
; rung 11: 12 - PROBLEMAS DE AQUECIMENTO
LD maq.def.def8
MOV(021) &12 maq.cparagem
; rung 12: 13 - FALHA DE SONDA
LD maq.cp_mes.cp13
MOV(021) &13 maq.cparagem
; rung 13: 15 - FUGA DE PRODUTO
LD maq.cp_mes.cp15
MOV(021) &15 maq.cparagem

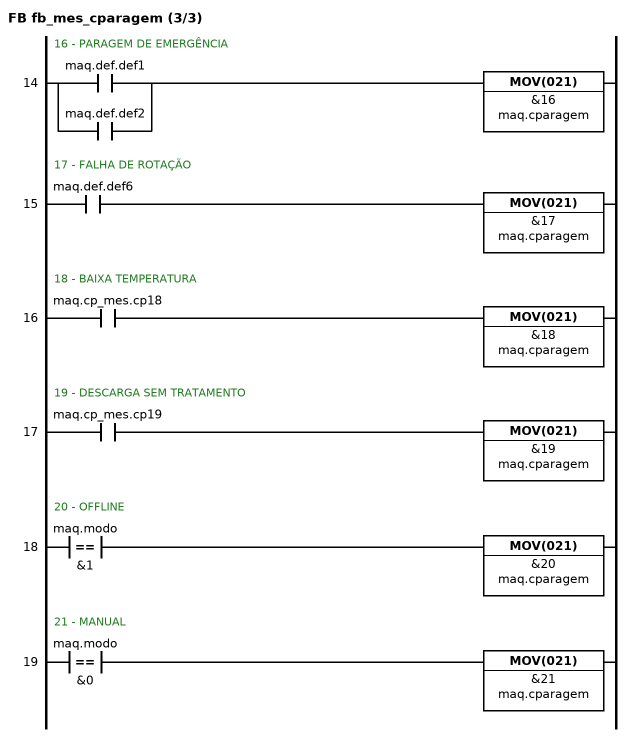
; rung 14: 16 - PARAGEM DE EMERGÊNCIA
LD maq.def.def1
OR maq.def.def2
MOV(021) &16 maq.cparagem
; rung 15: 17 - FALHA DE ROTAÇÃO
LD maq.def.def6
MOV(021) &17 maq.cparagem
; rung 16: 18 - BAIXA TEMPERATURA
LD maq.cp_mes.cp18
MOV(021) &18 maq.cparagem
; rung 17: 19 - DESCARGA SEM TRATAMENTO
LD maq.cp_mes.cp19
MOV(021) &19 maq.cparagem
; rung 18: 20 - OFFLINE
LD=(300) maq.modo &1
MOV(021) &20 maq.cparagem
; rung 19: 21 - MANUAL
LD=(300) maq.modo &0
MOV(021) &21 maq.cparagem

## Function block fb_of_clear
; FUNÇÃO LIMPA UMA ORDEM DE FABRICO - Coloca os valores da OF a zero.
VAR_IN_OUT
  of_in_out : s_of;  (* OF a ser apagada *)
END_VAR
(*Apaga uma OF*)
of_in_out.dados:= FALSE;

(*Cliente*)
of_in_out.cliente.nome[0]:=0;
of_in_out.cliente.nome[1]:=0;
of_in_out.cliente.nome[2]:=0;
of_in_out.cliente.nome[3]:=0;
of_in_out.cliente.nome[4]:=0;
of_in_out.cliente.nome[5]:=0;
of_in_out.cliente.nome[6]:=0;
of_in_out.cliente.nome[7]:=0;
of_in_out.cliente.nome[8]:=0;
of_in_out.cliente.nome[9]:=0;
of_in_out.cliente.nome[10]:=0;
of_in_out.cliente.nome[11]:=0;
of_in_out.cliente.nome[12]:=0;
of_in_out.cliente.nome[13]:=0;
of_in_out.cliente.nome[14]:=0;
of_in_out.cliente.nome[15]:=0;
of_in_out.cliente.nome[16]:=0;
of_in_out.cliente.nome[17]:=0;
of_in_out.cliente.nome[18]:=0;
of_in_out.cliente.nome[19]:=0;
of_in_out.cliente.nome[20]:=0;
of_in_out.cliente.nome[21]:=0;
of_in_out.cliente.nome[22]:=0;
of_in_out.cliente.nome[23]:=0;
of_in_out.cliente.nome[24]:=0;

of_in_out.cliente.data[0]:=0;
of_in_out.cliente.data[1]:=0;
of_in_out.cliente.data[2]:=0;
of_in_out.cliente.data[3]:=0;
of_in_out.cliente.data[4]:=0;
of_in_out.cliente.data[5]:=0;
of_in_out.cliente.data[6]:=0;
of_in_out.cliente.data[7]:=0;
of_in_out.cliente.data[8]:=0;
of_in_out.cliente.data[9]:=0;

of_in_out.cliente.produto[0]:=0;
of_in_out.cliente.produto[1]:=0;
of_in_out.cliente.produto[2]:=0;
of_in_out.cliente.produto[3]:=0;
of_in_out.cliente.produto[4]:=0;
of_in_out.cliente.produto[5]:=0;
of_in_out.cliente.produto[6]:=0;
of_in_out.cliente.produto[7]:=0;
of_in_out.cliente.produto[8]:=0;
of_in_out.cliente.produto[9]:=0;
of_in_out.cliente.produto[10]:=0;
of_in_out.cliente.produto[11]:=0;
of_in_out.cliente.produto[12]:=0;
of_in_out.cliente.produto[13]:=0;
of_in_out.cliente.produto[14]:=0;
of_in_out.cliente.produto[15]:=0;
of_in_out.cliente.produto[16]:=0;
of_in_out.cliente.produto[17]:=0;
of_in_out.cliente.produto[18]:=0;
of_in_out.cliente.produto[19]:=0;

of_in_out.cliente.prg_on[0]:=0;
of_in_out.cliente.prg_on[1]:=0;
of_in_out.cliente.prg_on[2]:=0;
of_in_out.cliente.prg_on[3]:=0;
of_in_out.cliente.prg_on[4]:=0;

of_in_out.cliente.n_enc[0]:=0;
of_in_out.cliente.n_enc[1]:=0;
of_in_out.cliente.n_enc[2]:=0;
of_in_out.cliente.n_enc[3]:=0;
of_in_out.cliente.n_enc[4]:=0;
of_in_out.cliente.n_enc[5]:=0;
of_in_out.cliente.n_enc[6]:=0;
of_in_out.cliente.n_enc[7]:=0;
of_in_out.cliente.n_enc[8]:=0;
of_in_out.cliente.n_enc[9]:=0;

of_in_out.cliente.n_of[0]:=0;
of_in_out.cliente.n_of[1]:=0;
of_in_out.cliente.n_of[2]:=0;
of_in_out.cliente.n_of[3]:=0;
of_in_out.cliente.n_of[4]:=0;
of_in_out.cliente.n_of[5]:=0;
of_in_out.cliente.n_of[6]:=0;
of_in_out.cliente.n_of[7]:=0;
of_in_out.cliente.n_of[8]:=0;
of_in_out.cliente.n_of[9]:=0;

of_in_out.cliente.n_lt[0]:=0;
of_in_out.cliente.n_lt[1]:=0;
of_in_out.cliente.n_lt[2]:=0;
of_in_out.cliente.n_lt[3]:=0;
of_in_out.cliente.n_lt[4]:=0;
of_in_out.cliente.n_lt[5]:=0;
of_in_out.cliente.n_lt[6]:=0;
of_in_out.cliente.n_lt[7]:=0;
of_in_out.cliente.n_lt[8]:=0;
of_in_out.cliente.n_lt[9]:=0;

(*Totais*)
of_in_out.totais.tt_global:=0;
of_in_out.totais.tt_falta:=0;
of_in_out.totais.tt_produzir:=0;

(*Calibre*)
of_in_out.calibre.dmt1:=0,0;
of_in_out.calibre.dmt2:=0,0;
of_in_out.calibre.h:=0,0;
of_in_out.calibre.a:=0,0;
of_in_out.calibre.qtp:=0,0;

of_in_out.calibre.cl_txt[0]:=0;
of_in_out.calibre.cl_txt[1]:=0;
of_in_out.calibre.cl_txt[2]:=0;
of_in_out.calibre.cl_txt[3]:=0;
of_in_out.calibre.cl_txt[4]:=0;
of_in_out.calibre.cl_txt[5]:=0;
of_in_out.calibre.cl_txt[6]:=0;
of_in_out.calibre.cl_txt[7]:=0;
of_in_out.calibre.cl_txt[8]:=0;
of_in_out.calibre.cl_txt[9]:=0;

(*Programa*)
of_in_out.prg.pss[0].f:=0;
of_in_out.prg.pss[0].p1:=0;
of_in_out.prg.pss[0].p2:=0,0;
of_in_out.prg.pss[0].tt:=0,0;
of_in_out.prg.pss[0].uni:=0;
of_in_out.prg.pss[0].uni:=12;
CASE of_in_out.prg.pss[0].f OF
	40:of_in_out.prg.pss[0].uni:=9;
END_CASE;

of_in_out.prg.pss[1].f:=0;
of_in_out.prg.pss[1].p1:=0;
of_in_out.prg.pss[1].p2:=0,0;
of_in_out.prg.pss[1].tt:=0,0;
of_in_out.prg.pss[1].uni:=0;
of_in_out.prg.pss[1].uni:=12;
CASE of_in_out.prg.pss[1].f OF
	40:of_in_out.prg.pss[1].uni:=9;
END_CASE;

of_in_out.prg.pss[2].f:=0;
of_in_out.prg.pss[2].p1:=0;
of_in_out.prg.pss[2].p2:=0,0;
of_in_out.prg.pss[2].tt:=0,0;
of_in_out.prg.pss[2].uni:=0;
of_in_out.prg.pss[2].uni:=12;
CASE of_in_out.prg.pss[2].f OF
	40:of_in_out.prg.pss[2].uni:=9;
END_CASE;

of_in_out.prg.pss[3].f:=0;
of_in_out.prg.pss[3].p1:=0;
of_in_out.prg.pss[3].p2:=0,0;
of_in_out.prg.pss[3].tt:=0,0;
of_in_out.prg.pss[3].uni:=0;
of_in_out.prg.pss[3].uni:=12;
CASE of_in_out.prg.pss[3].f OF
	40:of_in_out.prg.pss[3].uni:=9;
END_CASE;

of_in_out.prg.pss[4].f:=0;
of_in_out.prg.pss[4].p1:=0;
of_in_out.prg.pss[4].p2:=0,0;
of_in_out.prg.pss[4].tt:=0,0;
of_in_out.prg.pss[4].uni:=0;
of_in_out.prg.pss[4].uni:=12;
CASE of_in_out.prg.pss[4].f OF
	40:of_in_out.prg.pss[4].uni:=9;
END_CASE;

of_in_out.prg.pss[5].f:=0;
of_in_out.prg.pss[5].p1:=0;
of_in_out.prg.pss[5].p2:=0,0;
of_in_out.prg.pss[5].tt:=0,0;
of_in_out.prg.pss[5].uni:=0;
of_in_out.prg.pss[5].uni:=12;
CASE of_in_out.prg.pss[5].f OF
	40:of_in_out.prg.pss[5].uni:=9;
END_CASE;

of_in_out.prg.pss[6].f:=0;
of_in_out.prg.pss[6].p1:=0;
of_in_out.prg.pss[6].p2:=0,0;
of_in_out.prg.pss[6].tt:=0,0;
of_in_out.prg.pss[6].uni:=0;
of_in_out.prg.pss[6].uni:=12;
CASE of_in_out.prg.pss[6].f OF
	40:of_in_out.prg.pss[6].uni:=9;
END_CASE;

of_in_out.prg.pss[7].f:=0;
of_in_out.prg.pss[7].p1:=0;
of_in_out.prg.pss[7].p2:=0,0;
of_in_out.prg.pss[7].tt:=0,0;
of_in_out.prg.pss[7].uni:=0;
of_in_out.prg.pss[7].uni:=12;
CASE of_in_out.prg.pss[7].f OF
	40:of_in_out.prg.pss[7].uni:=9;
END_CASE;

of_in_out.prg.pss[8].f:=0;
of_in_out.prg.pss[8].p1:=0;
of_in_out.prg.pss[8].p2:=0,0;
of_in_out.prg.pss[8].tt:=0,0;
of_in_out.prg.pss[8].uni:=0;
of_in_out.prg.pss[8].uni:=12;
CASE of_in_out.prg.pss[8].f OF
	40:of_in_out.prg.pss[8].uni:=9;
END_CASE;

of_in_out.prg.pss[9].f:=0;
of_in_out.prg.pss[9].p1:=0;
of_in_out.prg.pss[9].p2:=0,0;
of_in_out.prg.pss[9].tt:=0,0;
of_in_out.prg.pss[9].uni:=0;
of_in_out.prg.pss[9].uni:=12;
CASE of_in_out.prg.pss[9].f OF
	40:of_in_out.prg.pss[9].uni:=9;
END_CASE;

of_in_out.prg.pss[10].f:=0;
of_in_out.prg.pss[10].p1:=0;
of_in_out.prg.pss[10].p2:=0,0;
of_in_out.prg.pss[10].tt:=0,0;
of_in_out.prg.pss[10].uni:=0;
of_in_out.prg.pss[10].uni:=12;
CASE of_in_out.prg.pss[10].f OF
	40:of_in_out.prg.pss[10].uni:=9;
END_CASE;

of_in_out.prg.pss[11].f:=0;
of_in_out.prg.pss[11].p1:=0;
of_in_out.prg.pss[11].p2:=0,0;
of_in_out.prg.pss[11].tt:=0,0;
of_in_out.prg.pss[11].uni:=0;
of_in_out.prg.pss[11].uni:=12;
CASE of_in_out.prg.pss[11].f OF
	40:of_in_out.prg.pss[11].uni:=9;
END_CASE;

## Function block fb_of_copy
; FUNÇÃO COPIA ORDENS DE FABRICO - Copia ordens de fabrico.
VAR_IN_OUT
  of_in : s_of;  (* OF original *)
  of_out : s_of;  (* OF para onde faz a copia *)
END_VAR
(*Copia de uma OF para outra*)
of_out.dados:=of_in.dados;

(*Cliente*)
of_out.cliente.nome[0]:=of_in.cliente.nome[0];
of_out.cliente.nome[1]:=of_in.cliente.nome[1];
of_out.cliente.nome[2]:=of_in.cliente.nome[2];
of_out.cliente.nome[3]:=of_in.cliente.nome[3];
of_out.cliente.nome[4]:=of_in.cliente.nome[4];
of_out.cliente.nome[5]:=of_in.cliente.nome[5];
of_out.cliente.nome[6]:=of_in.cliente.nome[6];
of_out.cliente.nome[7]:=of_in.cliente.nome[7];
of_out.cliente.nome[8]:=of_in.cliente.nome[8];
of_out.cliente.nome[9]:=of_in.cliente.nome[9];
of_out.cliente.nome[10]:=of_in.cliente.nome[10];
of_out.cliente.nome[11]:=of_in.cliente.nome[11];
of_out.cliente.nome[12]:=of_in.cliente.nome[12];
of_out.cliente.nome[13]:=of_in.cliente.nome[13];
of_out.cliente.nome[14]:=of_in.cliente.nome[14];
of_out.cliente.nome[15]:=of_in.cliente.nome[15];
of_out.cliente.nome[16]:=of_in.cliente.nome[16];
of_out.cliente.nome[17]:=of_in.cliente.nome[17];
of_out.cliente.nome[18]:=of_in.cliente.nome[18];
of_out.cliente.nome[19]:=of_in.cliente.nome[19];
of_out.cliente.nome[20]:=of_in.cliente.nome[20];
of_out.cliente.nome[21]:=of_in.cliente.nome[21];
of_out.cliente.nome[22]:=of_in.cliente.nome[22];
of_out.cliente.nome[23]:=of_in.cliente.nome[23];
of_out.cliente.nome[24]:=of_in.cliente.nome[24];

of_out.cliente.data[0]:=of_in.cliente.data[0];
of_out.cliente.data[1]:=of_in.cliente.data[1];
of_out.cliente.data[2]:=of_in.cliente.data[2];
of_out.cliente.data[3]:=of_in.cliente.data[3];
of_out.cliente.data[4]:=of_in.cliente.data[4];
of_out.cliente.data[5]:=of_in.cliente.data[5];
of_out.cliente.data[6]:=of_in.cliente.data[6];
of_out.cliente.data[7]:=of_in.cliente.data[7];
of_out.cliente.data[8]:=of_in.cliente.data[8];
of_out.cliente.data[9]:=of_in.cliente.data[9];

of_out.cliente.produto[0]:=of_in.cliente.produto[0];
of_out.cliente.produto[1]:=of_in.cliente.produto[1];
of_out.cliente.produto[2]:=of_in.cliente.produto[2];
of_out.cliente.produto[3]:=of_in.cliente.produto[3];
of_out.cliente.produto[4]:=of_in.cliente.produto[4];
of_out.cliente.produto[5]:=of_in.cliente.produto[5];
of_out.cliente.produto[6]:=of_in.cliente.produto[6];
of_out.cliente.produto[7]:=of_in.cliente.produto[7];
of_out.cliente.produto[8]:=of_in.cliente.produto[8];
of_out.cliente.produto[9]:=of_in.cliente.produto[9];
of_out.cliente.produto[10]:=of_in.cliente.produto[10];
of_out.cliente.produto[11]:=of_in.cliente.produto[11];
of_out.cliente.produto[12]:=of_in.cliente.produto[12];
of_out.cliente.produto[13]:=of_in.cliente.produto[13];
of_out.cliente.produto[14]:=of_in.cliente.produto[14];
of_out.cliente.produto[15]:=of_in.cliente.produto[15];
of_out.cliente.produto[16]:=of_in.cliente.produto[16];
of_out.cliente.produto[17]:=of_in.cliente.produto[17];
of_out.cliente.produto[18]:=of_in.cliente.produto[18];
of_out.cliente.produto[19]:=of_in.cliente.produto[19];

of_out.cliente.prg_on[0]:=of_in.cliente.prg_on[0];
of_out.cliente.prg_on[1]:=of_in.cliente.prg_on[1];
of_out.cliente.prg_on[2]:=of_in.cliente.prg_on[2];
of_out.cliente.prg_on[3]:=of_in.cliente.prg_on[3];
of_out.cliente.prg_on[4]:=of_in.cliente.prg_on[4];

of_out.cliente.n_enc[0]:=of_in.cliente.n_enc[0];
of_out.cliente.n_enc[1]:=of_in.cliente.n_enc[1];
of_out.cliente.n_enc[2]:=of_in.cliente.n_enc[2];
of_out.cliente.n_enc[3]:=of_in.cliente.n_enc[3];
of_out.cliente.n_enc[4]:=of_in.cliente.n_enc[4];
of_out.cliente.n_enc[5]:=of_in.cliente.n_enc[5];
of_out.cliente.n_enc[6]:=of_in.cliente.n_enc[6];
of_out.cliente.n_enc[7]:=of_in.cliente.n_enc[7];
of_out.cliente.n_enc[8]:=of_in.cliente.n_enc[8];
of_out.cliente.n_enc[9]:=of_in.cliente.n_enc[9];

of_out.cliente.n_of[0]:=of_in.cliente.n_of[0];
of_out.cliente.n_of[1]:=of_in.cliente.n_of[1];
of_out.cliente.n_of[2]:=of_in.cliente.n_of[2];
of_out.cliente.n_of[3]:=of_in.cliente.n_of[3];
of_out.cliente.n_of[4]:=of_in.cliente.n_of[4];
of_out.cliente.n_of[5]:=of_in.cliente.n_of[5];
of_out.cliente.n_of[6]:=of_in.cliente.n_of[6];
of_out.cliente.n_of[7]:=of_in.cliente.n_of[7];
of_out.cliente.n_of[8]:=of_in.cliente.n_of[8];
of_out.cliente.n_of[9]:=of_in.cliente.n_of[9];

of_out.cliente.n_lt[0]:=of_in.cliente.n_lt[0];
of_out.cliente.n_lt[1]:=of_in.cliente.n_lt[1];
of_out.cliente.n_lt[2]:=of_in.cliente.n_lt[2];
of_out.cliente.n_lt[3]:=of_in.cliente.n_lt[3];
of_out.cliente.n_lt[4]:=of_in.cliente.n_lt[4];
of_out.cliente.n_lt[5]:=of_in.cliente.n_lt[5];
of_out.cliente.n_lt[6]:=of_in.cliente.n_lt[6];
of_out.cliente.n_lt[7]:=of_in.cliente.n_lt[7];
of_out.cliente.n_lt[8]:=of_in.cliente.n_lt[8];
of_out.cliente.n_lt[9]:=of_in.cliente.n_lt[9];

(*Totais*)
of_out.totais.tt_global:=of_in.totais.tt_global;
of_out.totais.tt_falta:=of_in.totais.tt_falta;
of_out.totais.tt_produzir:=of_in.totais.tt_produzir;

(*Calibre*)
of_out.calibre.dmt1:=of_in.calibre.dmt1;
of_out.calibre.dmt2:=of_in.calibre.dmt2;
of_out.calibre.h:=of_in.calibre.h;
of_out.calibre.a:=of_in.calibre.a;
of_out.calibre.qtp:=of_in.calibre.qtp;

of_out.calibre.cl_txt[0]:= of_in.calibre.cl_txt[0];
of_out.calibre.cl_txt[1]:= of_in.calibre.cl_txt[1];
of_out.calibre.cl_txt[2]:= of_in.calibre.cl_txt[2];
of_out.calibre.cl_txt[3]:= of_in.calibre.cl_txt[3];
of_out.calibre.cl_txt[4]:= of_in.calibre.cl_txt[4];
of_out.calibre.cl_txt[5]:= of_in.calibre.cl_txt[5];
of_out.calibre.cl_txt[6]:= of_in.calibre.cl_txt[6];
of_out.calibre.cl_txt[7]:= of_in.calibre.cl_txt[7];
of_out.calibre.cl_txt[8]:= of_in.calibre.cl_txt[8];
of_out.calibre.cl_txt[9]:= of_in.calibre.cl_txt[9];

(*Programa*)
of_out.prg.pss[0].f:=of_in.prg.pss[0].f;
of_out.prg.pss[0].p1:=of_in.prg.pss[0].p1;
of_out.prg.pss[0].p2:=of_in.prg.pss[0].p2;
of_out.prg.pss[0].tt:=of_in.prg.pss[0].tt;
of_out.prg.pss[0].uni:=0;
of_out.prg.pss[0].uni:=12;
CASE of_out.prg.pss[0].f OF
	40:of_out.prg.pss[0].uni:=9;
END_CASE;

of_out.prg.pss[1].f:=of_in.prg.pss[1].f;
of_out.prg.pss[1].p1:=of_in.prg.pss[1].p1;
of_out.prg.pss[1].p2:=of_in.prg.pss[1].p2;
of_out.prg.pss[1].tt:=of_in.prg.pss[1].tt;
of_out.prg.pss[1].uni:=0;
of_out.prg.pss[1].uni:=12;
CASE of_out.prg.pss[1].f OF
	40:of_out.prg.pss[1].uni:=9;
END_CASE;

of_out.prg.pss[2].f:=of_in.prg.pss[2].f;
of_out.prg.pss[2].p1:=of_in.prg.pss[2].p1;
of_out.prg.pss[2].p2:=of_in.prg.pss[2].p2;
of_out.prg.pss[2].tt:=of_in.prg.pss[2].tt;
of_out.prg.pss[2].uni:=0;
of_out.prg.pss[2].uni:=12;
CASE of_out.prg.pss[2].f OF
	40:of_out.prg.pss[2].uni:=9;
END_CASE;

of_out.prg.pss[3].f:=of_in.prg.pss[3].f;
of_out.prg.pss[3].p1:=of_in.prg.pss[3].p1;
of_out.prg.pss[3].p2:=of_in.prg.pss[3].p2;
of_out.prg.pss[3].tt:=of_in.prg.pss[3].tt;
of_out.prg.pss[3].uni:=0;
of_out.prg.pss[3].uni:=12;
CASE of_out.prg.pss[3].f OF
	40:of_out.prg.pss[3].uni:=9;
END_CASE;

of_out.prg.pss[4].f:=of_in.prg.pss[4].f;
of_out.prg.pss[4].p1:=of_in.prg.pss[4].p1;
of_out.prg.pss[4].p2:=of_in.prg.pss[4].p2;
of_out.prg.pss[4].tt:=of_in.prg.pss[4].tt;
of_out.prg.pss[4].uni:=0;
of_out.prg.pss[4].uni:=12;
CASE of_out.prg.pss[4].f OF
	40:of_out.prg.pss[4].uni:=9;
END_CASE;

of_out.prg.pss[5].f:=of_in.prg.pss[5].f;
of_out.prg.pss[5].p1:=of_in.prg.pss[5].p1;
of_out.prg.pss[5].p2:=of_in.prg.pss[5].p2;
of_out.prg.pss[5].tt:=of_in.prg.pss[5].tt;
of_out.prg.pss[5].uni:=0;
of_out.prg.pss[5].uni:=12;
CASE of_out.prg.pss[5].f OF
	40:of_out.prg.pss[5].uni:=9;
END_CASE;

of_out.prg.pss[6].f:=of_in.prg.pss[6].f;
of_out.prg.pss[6].p1:=of_in.prg.pss[6].p1;
of_out.prg.pss[6].p2:=of_in.prg.pss[6].p2;
of_out.prg.pss[6].tt:=of_in.prg.pss[6].tt;
of_out.prg.pss[6].uni:=0;
of_out.prg.pss[6].uni:=12;
CASE of_out.prg.pss[6].f OF
	40:of_out.prg.pss[6].uni:=9;
END_CASE;

of_out.prg.pss[7].f:=of_in.prg.pss[7].f;
of_out.prg.pss[7].p1:=of_in.prg.pss[7].p1;
of_out.prg.pss[7].p2:=of_in.prg.pss[7].p2;
of_out.prg.pss[7].tt:=of_in.prg.pss[7].tt;
of_out.prg.pss[7].uni:=0;
of_out.prg.pss[7].uni:=12;
CASE of_out.prg.pss[7].f OF
	40:of_out.prg.pss[7].uni:=9;
END_CASE;

of_out.prg.pss[8].f:=of_in.prg.pss[8].f;
of_out.prg.pss[8].p1:=of_in.prg.pss[8].p1;
of_out.prg.pss[8].p2:=of_in.prg.pss[8].p2;
of_out.prg.pss[8].tt:=of_in.prg.pss[8].tt;
of_out.prg.pss[8].uni:=0;
of_out.prg.pss[8].uni:=12;
CASE of_out.prg.pss[8].f OF
	40:of_out.prg.pss[8].uni:=9;
END_CASE;

of_out.prg.pss[9].f:=of_in.prg.pss[9].f;
of_out.prg.pss[9].p1:=of_in.prg.pss[9].p1;
of_out.prg.pss[9].p2:=of_in.prg.pss[9].p2;
of_out.prg.pss[9].tt:=of_in.prg.pss[9].tt;
of_out.prg.pss[9].uni:=0;
of_out.prg.pss[9].uni:=12;
CASE of_out.prg.pss[9].f OF
	40:of_out.prg.pss[9].uni:=9;
END_CASE;

of_out.prg.pss[10].f:=of_in.prg.pss[10].f;
of_out.prg.pss[10].p1:=of_in.prg.pss[10].p1;
of_out.prg.pss[10].p2:=of_in.prg.pss[10].p2;
of_out.prg.pss[10].tt:=of_in.prg.pss[10].tt;
of_out.prg.pss[10].uni:=0;
of_out.prg.pss[10].uni:=12;
CASE of_out.prg.pss[10].f OF
	40:of_out.prg.pss[10].uni:=9;
END_CASE;

of_out.prg.pss[11].f:=of_in.prg.pss[11].f;
of_out.prg.pss[11].p1:=of_in.prg.pss[11].p1;
of_out.prg.pss[11].p2:=of_in.prg.pss[11].p2;
of_out.prg.pss[11].tt:=of_in.prg.pss[11].tt;
of_out.prg.pss[11].uni:=0;
of_out.prg.pss[11].uni:=12;
CASE of_out.prg.pss[11].f OF
	40:of_out.prg.pss[11].uni:=9;
END_CASE;

## Function block fb_of_copy_of_prg_prg
; FUNÇÃO COPIA PROGRAMA - Copia os 10 passos de um programa de uma OF para uma variavel do tipo PROGRAMA
VAR_IN_OUT
  in_of : s_of;  (* OF original *)
  out_prg : s_of_prg;  (* Programa para onde se faz a copia *)
END_VAR
(*Programa*)
out_prg.pss[0].f:=in_of.prg.pss[0].f;
out_prg.pss[0].p1:=in_of.prg.pss[0].p1;
out_prg.pss[0].p2:=in_of.prg.pss[0].p2;
out_prg.pss[0].tt:=in_of.prg.pss[0].tt;
out_prg.pss[0].uni:=in_of.prg.pss[0].uni;

out_prg.pss[1].f:=in_of.prg.pss[1].f;
out_prg.pss[1].p1:=in_of.prg.pss[1].p1;
out_prg.pss[1].p2:=in_of.prg.pss[1].p2;
out_prg.pss[1].tt:=in_of.prg.pss[1].tt;
out_prg.pss[1].uni:=in_of.prg.pss[1].uni;

out_prg.pss[2].f:=in_of.prg.pss[2].f;
out_prg.pss[2].p1:=in_of.prg.pss[2].p1;
out_prg.pss[2].p2:=in_of.prg.pss[2].p2;
out_prg.pss[2].tt:=in_of.prg.pss[2].tt;
out_prg.pss[2].uni:=in_of.prg.pss[2].uni;

out_prg.pss[3].f:=in_of.prg.pss[3].f;
out_prg.pss[3].p1:=in_of.prg.pss[3].p1;
out_prg.pss[3].p2:=in_of.prg.pss[3].p2;
out_prg.pss[3].tt:=in_of.prg.pss[3].tt;
out_prg.pss[3].uni:=in_of.prg.pss[3].uni;

out_prg.pss[4].f:=in_of.prg.pss[4].f;
out_prg.pss[4].p1:=in_of.prg.pss[4].p1;
out_prg.pss[4].p2:=in_of.prg.pss[4].p2;
out_prg.pss[4].tt:=in_of.prg.pss[4].tt;
out_prg.pss[4].uni:=in_of.prg.pss[4].uni;

out_prg.pss[5].f:=in_of.prg.pss[5].f;
out_prg.pss[5].p1:=in_of.prg.pss[5].p1;
out_prg.pss[5].p2:=in_of.prg.pss[5].p2;
out_prg.pss[5].tt:=in_of.prg.pss[5].tt;
out_prg.pss[5].uni:=in_of.prg.pss[5].uni;

out_prg.pss[6].f:=in_of.prg.pss[6].f;
out_prg.pss[6].p1:=in_of.prg.pss[6].p1;
out_prg.pss[6].p2:=in_of.prg.pss[6].p2;
out_prg.pss[6].tt:=in_of.prg.pss[6].tt;
out_prg.pss[6].uni:=in_of.prg.pss[6].uni;

out_prg.pss[7].f:=in_of.prg.pss[7].f;
out_prg.pss[7].p1:=in_of.prg.pss[7].p1;
out_prg.pss[7].p2:=in_of.prg.pss[7].p2;
out_prg.pss[7].tt:=in_of.prg.pss[7].tt;
out_prg.pss[7].uni:=in_of.prg.pss[7].uni;

out_prg.pss[8].f:=in_of.prg.pss[8].f;
out_prg.pss[8].p1:=in_of.prg.pss[8].p1;
out_prg.pss[8].p2:=in_of.prg.pss[8].p2;
out_prg.pss[8].tt:=in_of.prg.pss[8].tt;
out_prg.pss[8].uni:=in_of.prg.pss[8].uni;

out_prg.pss[9].f:=in_of.prg.pss[9].f;
out_prg.pss[9].p1:=in_of.prg.pss[9].p1;
out_prg.pss[9].p2:=in_of.prg.pss[9].p2;
out_prg.pss[9].tt:=in_of.prg.pss[9].tt;
out_prg.pss[9].uni:=in_of.prg.pss[9].uni;

out_prg.pss[10].f:=in_of.prg.pss[10].f;
out_prg.pss[10].p1:=in_of.prg.pss[10].p1;
out_prg.pss[10].p2:=in_of.prg.pss[10].p2;
out_prg.pss[10].tt:=in_of.prg.pss[10].tt;
out_prg.pss[10].uni:=in_of.prg.pss[10].uni;

out_prg.pss[11].f:=in_of.prg.pss[11].f;
out_prg.pss[11].p1:=in_of.prg.pss[11].p1;
out_prg.pss[11].p2:=in_of.prg.pss[11].p2;
out_prg.pss[11].tt:=in_of.prg.pss[11].tt;
out_prg.pss[11].uni:=in_of.prg.pss[11].uni;

## Function block fb_of_exe_calc
; FUNÇÃO CALCULO OF - Faz o escalonamento da OF para a dosagem especificada.
VAR_IN_OUT
  maq : s_maquina;  (* Dados da maquina *)
  of2_maq : s_of;  (* Dados da OF carregados na maquina *)
  prg_exe : s_of_prg;  (* Programa a executar *)
END_VAR
(* Calcula o programa*)
IF maq.bits.act_ciclo=FALSE AND maq.etapa<=20 THEN
	
	of2_maq.prg.pss[0].f:=prg_exe.pss[0].f;
	of2_maq.prg.pss[0].p1:=prg_exe.pss[0].p1;
	of2_maq.prg.pss[0].p2:=prg_exe.pss[0].p2;
	IF prg_exe.pss[0].f=40 THEN
		of2_maq.prg.pss[0].p2:= prg_exe.pss[0].p2*of2_maq.calibre.qtp/+100,0;
	END_IF;	
	of2_maq.prg.pss[0].tt:=prg_exe.pss[0].tt;
	of2_maq.prg.pss[0].uni:=prg_exe.pss[0].uni;
	
		
	of2_maq.prg.pss[1].f:=prg_exe.pss[1].f;
	of2_maq.prg.pss[1].p1:=prg_exe.pss[1].p1;
	of2_maq.prg.pss[1].p2:=prg_exe.pss[1].p2;
	IF prg_exe.pss[1].f=40 THEN
		of2_maq.prg.pss[1].p2:= prg_exe.pss[1].p2*of2_maq.calibre.qtp/+100,0;
	END_IF;	
	of2_maq.prg.pss[1].tt:=prg_exe.pss[1].tt;
	of2_maq.prg.pss[1].uni:=prg_exe.pss[1].uni;


	of2_maq.prg.pss[2].f:=prg_exe.pss[2].f;
	of2_maq.prg.pss[2].p1:=prg_exe.pss[2].p1;
	of2_maq.prg.pss[2].p2:=prg_exe.pss[2].p2;
	IF prg_exe.pss[2].f=40 THEN
		of2_maq.prg.pss[2].p2:= prg_exe.pss[2].p2*of2_maq.calibre.qtp/+100,0;
	END_IF;	
	of2_maq.prg.pss[2].tt:=prg_exe.pss[2].tt;
	of2_maq.prg.pss[2].uni:=prg_exe.pss[2].uni;


	of2_maq.prg.pss[3].f:=prg_exe.pss[3].f;
	of2_maq.prg.pss[3].p1:=prg_exe.pss[3].p1;
	of2_maq.prg.pss[3].p2:=prg_exe.pss[3].p2;
	IF prg_exe.pss[3].f=40 THEN
		of2_maq.prg.pss[3].p2:= prg_exe.pss[3].p2*of2_maq.calibre.qtp/+100,0;
	END_IF;	
	of2_maq.prg.pss[3].tt:=prg_exe.pss[3].tt;
	of2_maq.prg.pss[3].uni:=prg_exe.pss[3].uni;


	of2_maq.prg.pss[4].f:=prg_exe.pss[4].f;
	of2_maq.prg.pss[4].p1:=prg_exe.pss[4].p1;
	of2_maq.prg.pss[4].p2:=prg_exe.pss[4].p2;
	IF prg_exe.pss[4].f=40 THEN
		of2_maq.prg.pss[4].p2:= prg_exe.pss[4].p2*of2_maq.calibre.qtp/+100,0;
	END_IF;	
	of2_maq.prg.pss[4].tt:=prg_exe.pss[4].tt;
	of2_maq.prg.pss[4].uni:=prg_exe.pss[4].uni;


	of2_maq.prg.pss[5].f:=prg_exe.pss[5].f;
	of2_maq.prg.pss[5].p1:=prg_exe.pss[5].p1;
	of2_maq.prg.pss[5].p2:=prg_exe.pss[5].p2;
	IF prg_exe.pss[5].f=40 THEN
		of2_maq.prg.pss[5].p2:= prg_exe.pss[5].p2*of2_maq.calibre.qtp/+100,0;
	END_IF;	
	of2_maq.prg.pss[5].tt:=prg_exe.pss[5].tt;
	of2_maq.prg.pss[5].uni:=prg_exe.pss[5].uni;


	of2_maq.prg.pss[6].f:=prg_exe.pss[6].f;
	of2_maq.prg.pss[6].p1:=prg_exe.pss[6].p1;
	of2_maq.prg.pss[6].p2:=prg_exe.pss[6].p2;
	IF prg_exe.pss[6].f=40 THEN
		of2_maq.prg.pss[6].p2:= prg_exe.pss[6].p2*of2_maq.calibre.qtp/+100,0;
	END_IF;	
	of2_maq.prg.pss[6].tt:=prg_exe.pss[6].tt;
	of2_maq.prg.pss[6].uni:=prg_exe.pss[6].uni;


	of2_maq.prg.pss[7].f:=prg_exe.pss[7].f;
	of2_maq.prg.pss[7].p1:=prg_exe.pss[7].p1;
	of2_maq.prg.pss[7].p2:=prg_exe.pss[7].p2;
	IF prg_exe.pss[7].f=40 THEN
		of2_maq.prg.pss[7].p2:= prg_exe.pss[7].p2*of2_maq.calibre.qtp/+100,0;
	END_IF;	
	of2_maq.prg.pss[7].tt:=prg_exe.pss[7].tt;
	of2_maq.prg.pss[7].uni:=prg_exe.pss[7].uni;


	of2_maq.prg.pss[8].f:=prg_exe.pss[8].f;
	of2_maq.prg.pss[8].p1:=prg_exe.pss[8].p1;
	of2_maq.prg.pss[8].p2:=prg_exe.pss[8].p2;
	IF prg_exe.pss[8].f=40 THEN
		of2_maq.prg.pss[8].p2:= prg_exe.pss[8].p2*of2_maq.calibre.qtp/+100,0;
	END_IF;	
	of2_maq.prg.pss[8].tt:=prg_exe.pss[8].tt;
	of2_maq.prg.pss[8].uni:=prg_exe.pss[8].uni;


	of2_maq.prg.pss[9].f:=prg_exe.pss[9].f;
	of2_maq.prg.pss[9].p1:=prg_exe.pss[9].p1;
	of2_maq.prg.pss[9].p2:=prg_exe.pss[9].p2;
	IF prg_exe.pss[9].f=40 THEN
		of2_maq.prg.pss[9].p2:= prg_exe.pss[9].p2*of2_maq.calibre.qtp/+100,0;
	END_IF;	
	of2_maq.prg.pss[9].tt:=prg_exe.pss[9].tt;
	of2_maq.prg.pss[9].uni:=prg_exe.pss[9].uni;
	
	
	of2_maq.prg.pss[10].f:=prg_exe.pss[10].f;
	of2_maq.prg.pss[10].p1:=prg_exe.pss[10].p1;
	of2_maq.prg.pss[10].p2:=prg_exe.pss[10].p2;
	IF prg_exe.pss[10].f=40 THEN
		of2_maq.prg.pss[10].p2:= prg_exe.pss[10].p2*of2_maq.calibre.qtp/+100,0;
	END_IF;	
	of2_maq.prg.pss[10].tt:=prg_exe.pss[10].tt;
	of2_maq.prg.pss[10].uni:=prg_exe.pss[10].uni;
	
	
		of2_maq.prg.pss[11].f:=prg_exe.pss[11].f;
	of2_maq.prg.pss[11].p1:=prg_exe.pss[11].p1;
	of2_maq.prg.pss[11].p2:=prg_exe.pss[11].p2;
	IF prg_exe.pss[11].f=40 THEN
		of2_maq.prg.pss[11].p2:= prg_exe.pss[11].p2*of2_maq.calibre.qtp/+100,0;
	END_IF;	
	of2_maq.prg.pss[11].tt:=prg_exe.pss[11].tt;
	of2_maq.prg.pss[11].uni:=prg_exe.pss[11].uni;
	
END_IF;